// TIA Portal V17 export
// export: Created 2022-07-20T06:59:37.2106709Z, ExportSetting WithDefaults, DisplayName Totally Integrated Automation Portal, DisplayVersion V17, DisplayName TIA Portal Openness, DisplayVersion V17, DisplayName TIA Portal Version Control Interface, DisplayVersion V17, DisplayName SINAMICS Startdrive Advanced, DisplayVersion V17, DisplayName SINAMICS Startdrive G130, G150, S120, S150, SINAMICS MV, S210, DisplayVersion V17, DisplayName SINAMICS Startdrive G110M, G120, G120C, G120D, G120P, G115D, DisplayVersion V17, DisplayName STEP 7 Professional, DisplayVersion V17, DisplayName STEP 7 Safety, DisplayVersion V17, DisplayName WinCC Advanced, DisplayVersion V17
FUNCTION_BLOCK "FB10004_CheckPartnerAlive"   // FB10004, LAD
TITLE = FB10004_CheckPartnerAlive
{ S7_Optimized_Access := 'TRUE' }
AUTHOR : Anirouddh
FAMILY : 1000x_SYSTEM
VERSION : 1.0
// Release note : 
// 1.0 - Feature developped
// stored: AutoNumber false, IsIECCheckEnabled false, IsRetainMemResEnabled false, MemoryReserve 100, SetENOAutomatically false, UDAEnableTagReadback false
   VAR_INPUT
      KeepAliveSignal : UDInt;
      Acknowledge : Bool;
   END_VAR
   VAR_OUTPUT
      PartnerConnected : Bool;
      PartnerAlive : Bool;
   END_VAR
   VAR
      KeepAliveManagementStateDiagram : Int;
      NumberOfConsecutiveError : USInt;
      KeepAliveSignalTemp : UDInt;
      R_TRIG_PartnerAlive { S7_SetPoint := 'True'} : R_TRIG;
      R_TRIG_PartnerNotAlive { S7_SetPoint := 'True'} : R_TRIG;
      TON_Clock_200ms : TON_TIME;
   END_VAR
   VAR CONSTANT
      WAIT_FOR_PARTNER_CONNECTION : Int := 0;
      CONNEXION_RECORD_VALUE : Int := 10;
      CHECK_CONNEXION : Int := 20;
      ALIVE_RECORD_VALUE : Int := 30;
      CHECK_PARTNER_ALIVE : Int := 40;
   END_VAR
BEGIN

REGION Network 1 (SCL): FirstScan
   IF "FirstScan" THEN
       #PartnerAlive := FALSE;
       #PartnerConnected := FALSE;
       #KeepAliveSignalTemp := 0;
       #NumberOfConsecutiveError := 0;
       #KeepAliveManagementStateDiagram := #WAIT_FOR_PARTNER_CONNECTION;
   END_IF;
END_REGION

REGION Network 2 (SCL): Edge Signals & Timers
   REGION EDGE SIGNALS
   END_REGION

   REGION TIMERS    
       #TON_Clock_200ms(IN := #KeepAliveManagementStateDiagram = #CHECK_PARTNER_ALIVE,
                        PT := T#200ms);
   END_REGION
END_REGION

REGION Network 3 (SCL): Keep Alive Checking Management
   CASE #KeepAliveManagementStateDiagram OF
       #WAIT_FOR_PARTNER_CONNECTION:
           IF #KeepAliveSignal <> 0 THEN
               #KeepAliveManagementStateDiagram := #CONNEXION_RECORD_VALUE;
           END_IF;
       #CONNEXION_RECORD_VALUE:
           #KeepAliveSignalTemp := #KeepAliveSignal;
           #KeepAliveManagementStateDiagram := #CHECK_CONNEXION;
       #CHECK_CONNEXION:
           IF ABS(#KeepAliveSignalTemp - #KeepAliveSignal) > 50 THEN
               #PartnerConnected := TRUE;
               #KeepAliveManagementStateDiagram := #ALIVE_RECORD_VALUE;
           END_IF;
       #ALIVE_RECORD_VALUE:
           #KeepAliveSignalTemp := #KeepAliveSignal;
           #KeepAliveManagementStateDiagram := #CHECK_PARTNER_ALIVE;
       #CHECK_PARTNER_ALIVE:
           IF #TON_Clock_200ms.Q THEN
               IF #KeepAliveSignalTemp = #KeepAliveSignal THEN
                   #NumberOfConsecutiveError += 1;
               ELSE
                   #NumberOfConsecutiveError := 0;
                   #PartnerConnected := TRUE;
                   #PartnerAlive := TRUE;
               END_IF;
               RESET_TIMER(#TON_Clock_200ms);
               #KeepAliveManagementStateDiagram := #ALIVE_RECORD_VALUE;
           END_IF;
   END_CASE;
END_REGION

REGION Network 4 (SCL): Error Management
   IF #NumberOfConsecutiveError > 10 THEN
       #PartnerConnected := FALSE;
       #PartnerAlive := FALSE;
   ELSIF #Acknowledge THEN
       #KeepAliveManagementStateDiagram := #WAIT_FOR_PARTNER_CONNECTION;
       #NumberOfConsecutiveError := 0;
   END_IF;
END_REGION
END_FUNCTION_BLOCK
